FUNCTION_BLOCK CoE_property_string EXTENDS CoE_property
VAR_INPUT
END_VAR
VAR_OUTPUT
END_VAR
VAR
		_value : STRING;
END_VAR

SUPER^();

PROPERTY dataTypeSize : UINT
GET
dataTypeSize := SIZEOF(_value);
END_GET
END_PROPERTY

METHOD get_value : BOOL
VAR_OUTPUT
	value : STRING ;
	errId : UDINT;
END_VAR
IF init_done THEN
	value := _value;
	get_value := TRUE;
ELSE
	errId := 2;
	get_value := FALSE;
END_IF
END_METHOD

METHOD handle_read_callback : BOOL
VAR_INPUT
	pt_buffer : POINTER TO CoE_buffer_type_cast_union;
	errId : UDINT;
END_VAR

_value := pt_buffer^.value_string;
_init_done:=TRUE;
_read_errId:=errId;
END_METHOD

METHOD set_value : BOOL
VAR_INPUT
	value : string ;
END_VAR
_valueToWrite.value_string := value;
IF THIS^._CoE_property_handler <> 0 THEN 
	THIS^._CoE_property_handler.add_write_request(THIS^);
ELSE
	errId:=1;
END_IF
END_METHOD

END_FUNCTION_BLOCK

(* stored: Version 1.1.0.1, ProductVersion 3.1.4024.6
   POU CoE_property_string: Id {f55ea707-b327-0170-15c9-53696b6c1bbe}, SpecialFunc None
   Property dataTypeSize: Id {942166f3-1029-0217-1190-5fe89c28c610}
   Get Get: Id {f187cc8e-4648-0447-3b69-58389f3adfa9}
   Method get_value: Id {4daa8112-b93c-0b23-12a2-0debd286de3b}
   Method handle_read_callback: Id {33602f1a-b852-0193-2cb4-122fe6562bf0}
   Method set_value: Id {6a1d6304-dcc4-0939-23ae-bc7d895c061b} *)
